FUNCTION_BLOCK Throttle
  (* Standard: 61499-2 *)
  (* Version 0.2, 2003-12-04, JHC, Rockwell Automation, Renamed for better indexing. *)
  (* Version 0.1, 2002-11-05, JHC, Rockwell Automation, Corrected missing ST element in Algorithm REQ. *)
  (* Version 0.0, 2000-05-30, JHC, Rockwell Automation *)
  (* Compiler header: package fb.rt.benchmarks.cruisecontrol; *)
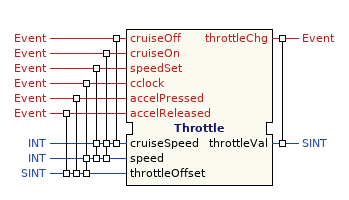
  EVENT_INPUT
    cruiseOff WITH cruiseSpeed;
    cruiseOn WITH cruiseSpeed, speed;
    speedSet WITH cruiseSpeed, speed;
    cclock WITH speed, throttleOffset; (* 10ms tick *)
    accelPressed WITH throttleOffset;
    accelReleased WITH throttleOffset;
  END_EVENT
  EVENT_OUTPUT
    throttleChg WITH throttleVal;
  END_EVENT
  VAR_INPUT
    cruiseSpeed : INT := 0; (* desired speed *)
    speed : INT := 0; (* actual speed *)
    throttleOffset : SINT := 0; (* offset angle *)
  END_VAR
  VAR_OUTPUT
    throttleVal : SINT := 0; (* throttle angle *)
  END_VAR
  VAR
    prevOffset : SINT := 0;
    tmp : SINT := 0;
  END_VAR
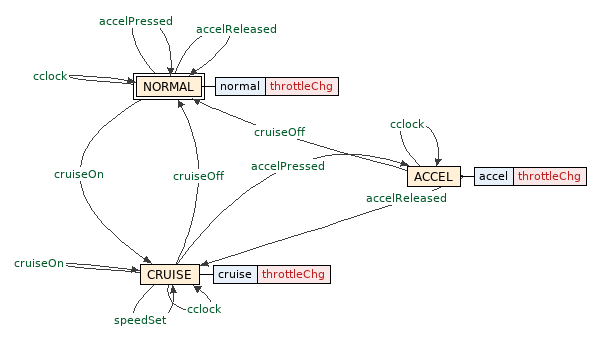
  EC_STATES
    NORMAL : normal -> throttleChg;
    CRUISE : cruise -> throttleChg;
    ACCEL : accel -> throttleChg;
  END_STATES
  EC_TRANSITIONS
    NORMAL TO CRUISE := cruiseOn;
    NORMAL TO NORMAL := accelPressed;
    NORMAL TO NORMAL := accelReleased;
    NORMAL TO NORMAL := cclock;
    CRUISE TO NORMAL := cruiseOff;
    CRUISE TO ACCEL := accelPressed;
    CRUISE TO CRUISE := cruiseOn;
    CRUISE TO CRUISE := speedSet;
    CRUISE TO CRUISE := cclock;
    ACCEL TO NORMAL := cruiseOff;
    ACCEL TO CRUISE := accelReleased;
    ACCEL TO ACCEL := cclock;
  END_TRANSITIONS
  ALGORITHM normal IN ST:
throttleVal := throttleOffset;
prevOffset := 0;
  END_ALGORITHM
  ALGORITHM accel IN ST:
throttleVal := throttleVal + throttleOffset - prevOffset;
prevOffset := throttleOffset;
  END_ALGORITHM
  ALGORITHM cruise IN ST:
tmp := (cruiseSpeed - speed);
tmp := tmp * 3;
 IF tmp > 45 THEN
    tmp := 45;
ELSIF tmp < 0 THEN
    tmp := 0;
 END_IF;
 throttleVal := tmp;
  END_ALGORITHM
END_FUNCTION_BLOCK
